# B&R Automation Studio project SuperTrakProject (part 2)

#### Main.st
```iecst
(***************************************************************************************
 * STSection task
 *
 * This task provides a state machine for controlling and monitoring
 * SuperTrak Sections. This task can be interfaced with via gSuperTrak.Sections
 *
 * File: STSection.st
 * Created: 2024-08-15
 *
 * Authors:
 *  Marcus Mangel, B&R Industrial Automation
 *  Tyler Matijevich, B&R Industrial Automation
 *
***************************************************************************************)

PROGRAM _CYCLIC

    // Read global inputs
    Interface.Cmd := gSuperTrak.Sections.Cmd;

    // Initialize common statuses, assume true/false then disqualify
    Interface.Status.Active := TRUE;
    Interface.Status.Error := FALSE;
	Interface.Status.SectionError := 0;
	Interface.Status.SectionWarning := 0;

    FOR Index := 1 TO ST_SECTION_MAX DO
        ControlSection[Index].StLink := ADR(gSTSystemLink);
        ControlSection[Index].Section := Index;
        // There are no function block parameters, use common address
        ControlSection[Index].Parameters := ADR(SectionParameters[Index]);
        // Enable all function blocks one the System is Active
        ControlSection[Index].Enable := gSuperTrak.System.Status.Active;
        // Enable each section
        ControlSection[Index].EnableSection := Interface.Cmd.PowerSection[Index] AND ControlSection[Index].MotorPowerOn AND NOT ControlSection[Index].Error;
        // Reset all function blocks
        ControlSection[Index].ErrorReset := gSuperTrak.System.Cmd.Reset AND ControlSection[Index].Error;
        ControlSection[Index]();

        // All sections must be active
        IF ControlSection[Index].Active = FALSE THEN
            Interface.Status.Active := FALSE;
        END_IF
        // Error if any section has error
        IF ControlSection[Index].Error THEN
            Interface.Status.Error := TRUE;
            Interface.Status.StatusID := ControlSection[Index].StatusID;
        END_IF
        IF ControlSection[Index].Info.SuperTrak.SectionFaultActive THEN
            Interface.Status.SectionError := Index;
		END_IF;
		IF ControlSection[Index].Info.SuperTrak.SectionWarningActive THEN
			Interface.Status.SectionWarning:= Index;
        END_IF;

        // Log errors only when that error first occurs
        r_trig_SectionFBError[Index](CLK := ControlSection[Index].Error);
        r_trig_SectionWarning[Index](CLK := ControlSection[Index].Info.SuperTrak.SectionWarningActive);
        r_trig_SectionFault[Index](CLK := ControlSection[Index].Info.SuperTrak.SectionFaultActive);

        IF r_trig_SectionFBError[Index].Q THEN
            brsmemset(ADR(UserLogArguments), 0, SIZEOF(UserLogArguments));
            UserLogArguments.i[0] := Index;
            UserLogArguments.i[1] := ControlSection[Index].StatusID;
            UserLogEventText('$$arlogusr', -536869812, 0, '', '%i %i', UserLogArguments);
        END_IF;
        IF r_trig_SectionWarning[Index].Q THEN
            brsmemset(ADR(UserLogArguments), 0, SIZEOF(UserLogArguments));
            UserLogArguments.i[0] := Index;
            UserLogArguments.i[1] := ControlSection[Index].Info.SuperTrak.SectionWarningBits;
            UserLogEventText('$$arlogusr', -1610609636, 0, '', '%i %i', UserLogArguments);
        END_IF;
        IF r_trig_SectionFault[Index].Q THEN
            brsmemset(ADR(UserLogArguments), 0, SIZEOF(UserLogArguments));
            UserLogArguments.i[0] := Index;
            UserLogArguments.i[1] := ControlSection[Index].Info.SuperTrak.SectionFaultBits;
            UserLogEventText('$$arlogusr', -536869810, 0, '', '%i %i', UserLogArguments);
        END_IF;

        // Read other statuses
        Interface.Info[Index].SectionEnabled := ControlSection[Index].SectionEnabled;
        Interface.Info[Index].UnrecognizedShuttles := ControlSection[Index].UnrecognizedPallets;
        Interface.Info[Index].MotorPowerOn := ControlSection[Index].MotorPowerOn;
        Interface.Info[Index].ShuttlesRecovering := ControlSection[Index].PalletsRecovering;
        Interface.Info[Index].LocatingShuttles := ControlSection[Index].LocatingPallets;
        Interface.Info[Index].DisabledExternally := ControlSection[Index].DisabledExternally;
        Interface.Info[Index].WarningPresent := ControlSection[Index].Info.SuperTrak.SectionWarningActive;
        Interface.Info[Index].Warnings := ControlSection[Index].Info.SuperTrak.SectionWarningBits;
        Interface.Info[Index].FaultPresent := ControlSection[Index].Info.SuperTrak.SectionFaultActive;
        Interface.Info[Index].Faults := ControlSection[Index].Info.SuperTrak.SectionFaultBits;
    END_FOR

    // Write global outputs
	gSuperTrak.Sections.Status := Interface.Status;
	gSuperTrak.Sections.Info := Interface.Info;

END_PROGRAM
```

### Package Logical/Source/STMgr/STTarget - StCom target control

### STTarget.typ - Global types
```iecst
(***************************************************************************************
 * Global STTarget data types
 *
 * These structures allow any program (task) to interface with the STTarget task
 *
 * File: STTarget.typ
 * Created: 2024-08-15
 *
 * Authors:
 *  Marcus Mangel, B&R Industrial Automation
 *
****************************************************************************************)

TYPE
    STTargetInterfaceType :     STRUCT  (*Target control interface*)
        Cmd : STTargetCommandType; (*Target release and set shuttle parameter commands*)
        Par : STTargetParType; (*Target control parameters*)
        Status : STTargetStatusType; (*Target status structure*)
    END_STRUCT;
    STTargetCommandType :     STRUCT  (*Target release and set shuttle parameter commands*)
        Release : STReleaseCommandType; (*Target release commands*)
        SetShuttleID : BOOL; (*Set the ID of the shuttle at the target*)
    END_STRUCT;
    STTargetParType :     STRUCT  (*Target control parameters*)
        Release : STReleaseParameterType; (*Target release parameters*)
        SetShuttleID : USINT; (*Set the current shuttle's ID to this when commanded*)
    END_STRUCT;
    STTargetStatusType :     STRUCT  (*Target status structure*)
        Active : BOOL; (*Target Control function block is active*)
        Error : BOOL; (*Target Control function block is reporting an error*)
        StatusID : DINT; (*Status ID from the Target Control function block*)
        ShuttlePresent : BOOL; (*A shuttle has arrived, has entered the in-position window, and has not yet been released*)
        ShuttleInPosition : BOOL; (*A shuttle is currently within the in-position window*)
        ShuttlePreArrival : BOOL; (*A shuttle is expected to arrive at the stop within the configured time*)
        ShuttleOverTarget : BOOL; (*A shuttle's shelf is over the target, only reported if configured*)
        ShuttleOffsetIndex : USINT; (*Offset-Table index applied to the shuttle at the target*)
        ShuttleID : USINT; (*ID of shuttle present at target, pallet over target (if configured), or pallet from pre-arrival notification (if configured)*)
        ShuttleReleased : BOOL; (*(Derived) Release command acknowledged. True until release command is reset*)
        ShuttleCount : USINT; (*(Derived) Number of shuttles destined for target*)
        Section : USINT; (*(Par 1650) Target section number*)
        PositionMicrons : DINT; (*(Par 1651) [um] Target section position in microns*)
        Position : REAL; (*(Par 1651) [mm] Target section position*)
        ShuttleIDSet : BOOL; (*The Shuttle ID was successfully set. True until the command is reset*)
    END_STRUCT;
END_TYPE
```

### Program Logical/Source/STMgr/STTarget/STTarget (IEC) - StCom target control

#### Main.st - Init, cyclic, exit code
```iecst
(***************************************************************************************
 * STTarget task
 *
 * This task provides a state machine for controlling and monitoring
 * SuperTrak Targets. This task can be interfaced with via gSuperTrak.Target[Target #]
 * where "Target #" is an array value indexed starting at 1 (see: Trakmaster targets)
 *
 * File: STTarget.st
 * Created: 2024-08-15
 *
 * Authors:
 *  Marcus Mangel, B&R Industrial Automation
 *
***************************************************************************************)

PROGRAM _CYCLIC

    // Get data for all targets when the system is active
    IF gSuperTrak.System.Status.Active THEN
        SuperTrakServChanRead(0, 1650, 0, 256, ADR(Sections), SIZEOF(Sections));
        SuperTrakServChanRead(0, 1651, 0, 256, ADR(Positions), SIZEOF(Positions));
    END_IF;

    FOR Index := 1 TO ST_TARGET_MAX DO
        // Read global inputs
        Interface[Index].Cmd := gSuperTrak.Target[Index].Cmd;
        Interface[Index].Par := gSuperTrak.Target[Index].Par;

        // Link parameters
        TargetParameters[Index].AdvancedReleaseConfig.DestinationTarget := Interface[Index].Par.Release.DestinationTarget;
        TargetParameters[Index].AdvancedReleaseConfig.IncrementalOffset := LIMIT(-500.0, Interface[Index].Par.Release.IncrementalOffset, 500.0);
        TargetParameters[Index].AdvancedReleaseConfig.TargetOffset := LIMIT(-500.0, Interface[Index].Par.Release.TargetOffset, 500.0);
        TargetParameters[Index].AdvancedReleaseConfig.Direction := Interface[Index].Par.Release.Direction;
        TargetParameters[Index].PalletConfig.Motion.Acceleration := REAL_TO_UINT(LIMIT(1, Interface[Index].Par.Release.Acceleration, 60) * METERS_TO_MILLIMETERS);
        TargetParameters[Index].PalletConfig.Motion.Velocity := REAL_TO_UINT(LIMIT(10, Interface[Index].Par.Release.Velocity, 4000));
        TargetParameters[Index].PalletConfig.ID := Interface[Index].Par.SetShuttleID;

        // StTargetExt function block inputs
        ControlTarget[Index].StLink := ADR(gSTSystemLink);
        ControlTarget[Index].Enable := gSuperTrak.System.Status.Active;
        ControlTarget[Index].ErrorReset := gSuperTrak.System.Cmd.Reset AND ControlTarget[Index].Error;
        ControlTarget[Index].Parameters := ADR(TargetParameters[Index]);
        ControlTarget[Index].Target := Index;

        // If the function block errored out, reset it's commands to prevent an error loop
        IF ControlTarget[Index].ErrorReset THEN
            ControlTarget[Index].ReleaseToTarget := FALSE;
            ControlTarget[Index].ReleaseToOffset := FALSE;
            ControlTarget[Index].IncrementOffset := FALSE;
	        TargetControlState[Index] := TARGET_STATE_WAIT_FOR_CMD_RESET;
        END_IF;

        CASE TargetControlState[Index] OF
            TARGET_STATE_WAIT_FOR_SHUTTLE:
                IF ControlTarget[Index].PalletPresent THEN
                    TargetControlState[Index] := TARGET_STATE_SHUTTLE_PRESENT;
                END_IF;

            TARGET_STATE_SHUTTLE_PRESENT:
                IF Interface[Index].Cmd.SetShuttleID THEN
                    TargetControlState[Index] := TARGET_STATE_SET_SHUTTLE_ID;
                ELSIF Interface[Index].Cmd.Release.ReleaseToTarget OR Interface[Index].Cmd.Release.ReleaseToOffset OR Interface[Index].Cmd.Release.IncrementOffset THEN
                    TargetControlState[Index] := TARGET_STATE_SET_MOTION_PARS;
                END_IF;

            TARGET_STATE_SET_SHUTTLE_ID:
                ControlTarget[Index].SetPalletID := TRUE;
                IF ControlTarget[Index].CommandDone THEN
                    ControlTarget[Index].SetPalletID := FALSE;
                    Interface[Index].Status.ShuttleIDSet := TRUE;
                    TargetControlState[Index] := TARGET_STATE_WAIT_FOR_CMD_RESET;
                END_IF;

            TARGET_STATE_SET_MOTION_PARS:
                ControlTarget[Index].SetPalletMotionPar := TRUE;
                IF ControlTarget[Index].CommandDone THEN
                    ControlTarget[Index].SetPalletMotionPar := FALSE;
                    TargetControlState[Index] := TARGET_STATE_RELEASE_SHUTTLE;
                END_IF;

            TARGET_STATE_RELEASE_SHUTTLE:
                ControlTarget[Index].ReleaseToTarget := Interface[Index].Cmd.Release.ReleaseToTarget; // Trust that the user won't set more than
                ControlTarget[Index].ReleaseToOffset := Interface[Index].Cmd.Release.ReleaseToOffset; // one of these at the same time
                ControlTarget[Index].IncrementOffset := Interface[Index].Cmd.Release.IncrementOffset; // Not sure what would happen in that case
                TargetControlState[Index] := TARGET_STATE_WAIT_FOR_RELEASE;

            TARGET_STATE_WAIT_FOR_RELEASE:
                IF NOT ControlTarget[Index].PalletPresent THEN
                    ControlTarget[Index].ReleaseToTarget := FALSE;
                    ControlTarget[Index].ReleaseToOffset := FALSE;
                    ControlTarget[Index].IncrementOffset := FALSE;
                    Interface[Index].Status.ShuttleReleased := TRUE;
                    TargetControlState[Index] := TARGET_STATE_WAIT_FOR_CMD_RESET;
                END_IF;

            TARGET_STATE_WAIT_FOR_CMD_RESET:
                IF NOT (Interface[Index].Cmd.SetShuttleID OR Interface[Index].Cmd.Release.ReleaseToTarget
                    OR Interface[Index].Cmd.Release.ReleaseToOffset OR Interface[Index].Cmd.Release.IncrementOffset) THEN
                    Interface[Index].Status.ShuttleReleased := FALSE;
                    Interface[Index].Status.ShuttleIDSet := FALSE; // Reset all "Command Done" Statuses
                    TargetControlState[Index] := TARGET_STATE_WAIT_FOR_SHUTTLE;
                END_IF;
        END_CASE;

        // Call StTargetExt function block
        ControlTarget[Index]();

        // Read StTargetExt function block outputs
        Interface[Index].Status.Active := ControlTarget[Index].Active;
        Interface[Index].Status.Error := ControlTarget[Index].Error;
        Interface[Index].Status.StatusID := ControlTarget[Index].StatusID;
        Interface[Index].Status.ShuttleID := ControlTarget[Index].PalletID;
        Interface[Index].Status.ShuttleOffsetIndex := ControlTarget[Index].PalletOffsetIdx;
        Interface[Index].Status.ShuttlePresent := ControlTarget[Index].PalletPresent;
        Interface[Index].Status.ShuttleInPosition := ControlTarget[Index].PalletInPosition;
        Interface[Index].Status.ShuttlePreArrival := ControlTarget[Index].PalletPreArrival;
        Interface[Index].Status.ShuttleOverTarget := ControlTarget[Index].PalletOverTarget;
        Interface[Index].Status.Section := UINT_TO_USINT(Sections[Index]);
        Interface[Index].Status.PositionMicrons := Positions[Index];
        Interface[Index].Status.Position := DINT_TO_REAL(Interface[Index].Status.PositionMicrons)/1000.0;

        // Log errors only when that error first occurs
        r_trig_TargetFBError[Index](CLK := ControlTarget[Index].Error);

        IF r_trig_TargetFBError[Index].Q THEN
            brsmemset(ADR(UserLogArguments), 0, SIZEOF(UserLogArguments));
            UserLogArguments.i[0] := Index;
            UserLogArguments.i[1] := ControlTarget[Index].StatusID;
            UserLogEventText('$$arlogusr', -536869712, 0, '', '%i %i', UserLogArguments);
        END_IF;

        // Check for release commands and update ShuttleCount status
        r_trig_ShuttleRelease[Index].CLK := (Interface[Index].Cmd.Release.ReleaseToTarget
        OR Interface[Index].Cmd.Release.ReleaseToOffset OR Interface[Index].Cmd.Release.IncrementOffset);
        r_trig_ShuttleRelease[Index]();

        IF r_trig_ShuttleRelease[Index].Q THEN
            // Decrement this target's shuttle count
            IF Interface[Index].Status.ShuttleCount > 0 THEN
                Interface[Index].Status.ShuttleCount := Interface[Index].Status.ShuttleCount - 1;
            END_IF;
            // Increment destination target's shuttle count
            IF Interface[Index].Par.Release.DestinationTarget > 0 AND Interface[Index].Par.Release.DestinationTarget <= ST_TARGET_MAX THEN
                Interface[Interface[Index].Par.Release.DestinationTarget].Status.ShuttleCount :=
                Interface[Interface[Index].Par.Release.DestinationTarget].Status.ShuttleCount + 1;
            END_IF;
        END_IF;

        // Write global outputs
        gSuperTrak.Target[Index].Status := Interface[Index].Status;
    END_FOR

END_PROGRAM
```

#### Types.typ
```iecst
(***************************************************************************************
 * STTarget task local data types
 *
 * These structures and enumerations are local to the STTarget task
 *
 * File: STTarget/Types.typ
 * Created: 2024-08-15
 *
 * Authors:
 *  Marcus Mangel, B&R Industrial Automation
 *
***************************************************************************************)
TYPE
	TargetControlState_enum :
		( (*Shuttle release state machine*)
		TARGET_STATE_WAIT_FOR_SHUTTLE, (*Wait for a shuttle to arrive at the target*)
		TARGET_STATE_SHUTTLE_PRESENT, (*A shuttle is at the target and ready for commands*)
		TARGET_STATE_SET_SHUTTLE_ID, (*Set the ID of the shuttle that is currently at the target*)
		TARGET_STATE_SET_MOTION_PARS, (*Set the shutte at target's motion parameters*)
		TARGET_STATE_RELEASE_SHUTTLE, (*Release the shuttle currently at the target*)
		TARGET_STATE_WAIT_FOR_RELEASE, (*Wait for the release to complete*)
		TARGET_STATE_WAIT_FOR_CMD_RESET (*Wait for the caller to reset all commands*)
		);
END_TYPE
```

#### Variables.var - Local variables
```iecst
(***************************************************************************************
 * STTarget task local variables
 *
 * These variables are local to the STTarget task
 *
 * File: STTarget/Variables.var
 * Created: 2024-08-15
 *
 * Authors:
 *  Marcus Mangel, B&R Industrial Automation
 *
***************************************************************************************)
VAR
	Interface : ARRAY[1..ST_TARGET_MAX] OF STTargetInterfaceType; (*Local copy of gSuperTrak.Target*)
	TargetControlState : ARRAY[1..ST_TARGET_MAX] OF TargetControlState_enum; (*Shuttle release state machine*)
	TargetParameters : ARRAY[1..ST_TARGET_MAX] OF StTargetExtParType; (*Target control parameters*)
	ControlTarget : ARRAY[1..ST_TARGET_MAX] OF StTargetExt; (*Target control function block*)
	Sections : ARRAY[0..255] OF UINT; (*All target sections*)
	Positions : ARRAY[0..255] OF DINT; (*All target positions*)
	Index : USINT; (*FOR loop index*)
	r_trig_ShuttleRelease : ARRAY[1..ST_TARGET_MAX] OF R_TRIG; (*Rising edge trigger of any Release command*)
	UserLogArguments : UserLogFormatType; (*Arguments used in Logger messages (UserLog library)*)
	r_trig_TargetFBError : ARRAY[1..ST_TARGET_MAX] OF R_TRIG; (*Rising edge trigger for ControlTarget.Error*)
END_VAR
```

### Package Logical/Source/STMgr/STShuttle - StCom shuttle (pallet) control

### STShuttle.typ - Global types
```iecst
(***************************************************************************************
 * Global STShuttle data types
 *
 * These structures allow any program (task) to interface with the STShuttle task
 *
 * File: STShuttle.typ
 * Created: 2024-08-15
 *
 * Authors:
 *  Marcus Mangel, B&R Industrial Automation
 *
****************************************************************************************)

TYPE
    STShuttleInterfaceType :     STRUCT  (*Shuttle interface structure*)
        Cmd : STReleaseCommandType; (*Shuttle release commands*)
        Status : STShuttleStatusType; (*Shuttle status information*)
        Par : STReleaseParameterType; (*Shuttle release parameters*)
    END_STRUCT;
    STShuttleStatusType :     STRUCT  (*Shuttle status structure*)
        Active : BOOL; (*Shuttle Control function block is active*)
        Error : BOOL; (*Shuttle Control function block is reporting an error*)
        StatusID : DINT; (*Status ID from the Shuttle Control function block*)
        ShuttleID : USINT; (*(StPalletStatusBits_e) ID Number assigned to the shuttle*)
        Present : BOOL; (*(StPalletStatusBits_e) Present on system*)
        Recovering : BOOL; (*(StPalletStatusBits_e) Will recover or recovering to last controlled position*)
        AtTarget : BOOL; (*(StPalletStatusBits_e) Arrived at target, in position, not yet released*)
        InPosition : BOOL; (*(StPalletStatusBits_e) Within in-position window*)
        ServoEnabled : BOOL; (*(StPalletStatusBits_e) Control enabled*)
        Initializing : BOOL; (*(StPalletStatusBits_e) Moving to load target*)
        Lost : BOOL; (*(StPalletStatusBits_e) Position feedback lost*)
        ControlMode : USINT; (*(SuperTrakPalletInfo_t) Pallet control mode, see SuperTrak library*)
        Section : USINT; (*(SuperTrakPalletInfo_t or Par 1307) Current section number*)
        PositionMicrons : DINT; (*(SuperTrakPalletInfo_t or Par 1310) [um] Current section position in microns*)
        Position : REAL; (*(SuperTrakPalletInfo_t or Par 1310) [mm] Current section position*)
        Velocity : REAL; (*(Par 1314) [mm/s] Current velocity*)
        DestinationTarget : USINT; (*(Par 1339) Destination target*)
        SetSection : USINT; (*(Par 1306) Section number setpoint*)
        SetPositionMicrons : DINT; (*(Par 1311) [um] Integer section position setpoint in microns*)
        SetPosition : REAL; (*(Par 1311) [mm] Section position setpoint*)
        SetVelocity : REAL; (*(Par 1313) [mm/s] Velocity setpoint*)
        SetAcceleration : REAL; (*(Par 1312) [m/s^2] Acceleration setpoint (raw value is mm/s^2!]*)
        ShuttleReleased : BOOL; (*(Derived) Release command acknowledged. True until release command is reset*)
    END_STRUCT;
END_TYPE
```

### Program Logical/Source/STMgr/STShuttle/STShuttle (IEC) - StCom shuttle control

#### Types.typ
```iecst
(***************************************************************************************
 * STShuttle task local data types
 *
 * These structures and enumerations are local to the STShuttle task
 *
 * File: STShuttle/Types.typ
 * Created: 2024-08-15
 *
 * Authors:
 *  Marcus Mangel, B&R Industrial Automation
 *
***************************************************************************************)
TYPE
	ShuttleControlState_enum :
		( (*State machine for Shuttle control*)
		SHUTTLE_STATE_WAIT_FOR_COMMAND, (*Wait for a command*)
		SHUTTLE_STATE_SET_MOTION_PARS, (*Set the shuttle's velocity and acceleration*)
		SHUTTLE_STATE_RELEASE_SHUTTLE, (*Give the shuttle a release command*)
		SHUTTLE_STATE_WAIT_FOR_CMD_RESET (*Wait for interface commands to be reset by the caller*)
		);
END_TYPE
```

#### Variables.var
```iecst
(***************************************************************************************
 * STShuttle task local variables
 *
 * These variables are local to the STShuttle task
 *
 * File: STShuttle/Variables.var
 * Created: 2024-08-15
 *
 * Authors:
 *  Marcus Mangel, B&R Industrial Automation
 *
***************************************************************************************)
VAR
	Interface : ARRAY[1..ST_SHUTTLE_MAX] OF STShuttleInterfaceType; (*Local copy of gSuperTrak.Shuttle*)
	ShuttleControlState : ARRAY[1..ST_SHUTTLE_MAX] OF ShuttleControlState_enum; (*Shuttle release state machine*)
	ShuttleParameters : ARRAY[1..ST_SHUTTLE_MAX] OF StPalletParType; (*Shuttle control parameters*)
	ControlShuttle : ARRAY[1..ST_SHUTTLE_MAX] OF StPallet; (*Shuttle control function block*)
	ShuttleInfo : ARRAY[1..ST_SHUTTLE_MAX] OF SuperTrakPalletInfo_t; (*Shuttle status information*)
	ActualVelocity : ARRAY[0..255] OF INT; (*Actual Velocity information for all shuttles*)
	DestinationTarget : ARRAY[0..255] OF UINT; (*Destination Target information for all shuttles*)
	SectionSetpoint : ARRAY[0..255] OF UINT; (*Section Setpoint information for all shuttles*)
	PositionSetpoint : ARRAY[0..255] OF DINT; (*Position Setpoint information for all shuttles*)
	VelocitySetpoint : ARRAY[0..255] OF REAL; (*Velocity Setpoint information for all shuttles*)
	AccelerationSetpoint : ARRAY[0..255] OF REAL; (*Acceleration Setpoint information for all shuttles*)
	Index : USINT; (*FOR Loop index*)
	r_trig_ShuttleRelease : ARRAY[1..ST_SHUTTLE_MAX] OF R_TRIG; (*Rising edge trigger of any Release command*)
	ShuttleAtTarget : USINT; (*Used during release to check the Target a Shuttle is currently at*)
	TargetIndex : USINT; (*FOR loop index*)
	UserLogArguments : UserLogFormatType; (*Arguments used in Logger messages (UserLog library)*)
	r_trig_ShuttleFBError : ARRAY[1..ST_SHUTTLE_MAX] OF R_TRIG; (*Rising edge trigger for ControlShuttle.Error*)
END_VAR
```

#### Main.st
```iecst
(*******************************************************************************************
 * STShuttle task
 *
 * This task provides a state machine for controlling and monitoring
 * SuperTrak Shuttles. This task can be interfaced with via gSuperTrak.Shuttle[Shuttle #]
 * where "Shuttle #" is an array value indexed starting at 1 (see: Trakmaster shuttles)
 *
 * File: STShuttle.st
 * Created: 2024-08-15
 *
 * Authors:
 *  Marcus Mangel, B&R Industrial Automation
 *
*******************************************************************************************)

PROGRAM _CYCLIC

    // Get data for all shuttles when the system is active
    IF gSuperTrak.System.Status.Active THEN
        // Call SuperTrakGetPalletInfo function
        SuperTrakGetPalletInfo(ADR(ShuttleInfo), SIZEOF(ShuttleInfo)/SIZEOF(ShuttleInfo[1]), FALSE); // FALSE - Return actual positions of shuttles

        // Read additional parameters via the Service Channel
        SuperTrakServChanRead(0, 1314, 0, 256, ADR(ActualVelocity), SIZEOF(ActualVelocity));
        SuperTrakServChanRead(0, 1339, 0, 256, ADR(DestinationTarget), SIZEOF(DestinationTarget));
        SuperTrakServChanRead(0, 1306, 0, 256, ADR(SectionSetpoint), SIZEOF(SectionSetpoint));
        SuperTrakServChanRead(0, 1311, 0, 256, ADR(PositionSetpoint), SIZEOF(PositionSetpoint));
        SuperTrakServChanRead(0, 1313, 0, 256, ADR(VelocitySetpoint), SIZEOF(VelocitySetpoint));
        SuperTrakServChanRead(0, 1312, 0, 256, ADR(AccelerationSetpoint), SIZEOF(AccelerationSetpoint));
    END_IF;

    FOR Index := 1 TO ST_SHUTTLE_MAX DO
        // Read global inputs
        Interface[Index].Cmd := gSuperTrak.Shuttle[Index].Cmd;
        Interface[Index].Par := gSuperTrak.Shuttle[Index].Par;

        // Link parameters
        ShuttleParameters[Index].AdvancedReleaseConfig.DestinationTarget := Interface[Index].Par.DestinationTarget;
        ShuttleParameters[Index].AdvancedReleaseConfig.IncrementalOffset := LIMIT(-500.0, Interface[Index].Par.IncrementalOffset, 500.0);
        ShuttleParameters[Index].AdvancedReleaseConfig.TargetOffset := LIMIT(-500.0, Interface[Index].Par.TargetOffset, 500.0);
        ShuttleParameters[Index].AdvancedReleaseConfig.Direction := Interface[Index].Par.Direction;
        ShuttleParameters[Index].PalletConfig.Motion.Acceleration := REAL_TO_UINT(LIMIT(1, Interface[Index].Par.Acceleration, 60) * METERS_TO_MILLIMETERS);
        ShuttleParameters[Index].PalletConfig.Motion.Velocity := REAL_TO_UINT(LIMIT(10, Interface[Index].Par.Velocity, 4000));

        // StShuttleExt function block inputs
        ControlShuttle[Index].StLink := ADR(gSTSystemLink);
        ControlShuttle[Index].Enable := gSuperTrak.System.Status.Active;
        ControlShuttle[Index].ErrorReset := gSuperTrak.System.Cmd.Reset AND ControlShuttle[Index].Error;
        ControlShuttle[Index].Parameters := ADR(ShuttleParameters[Index]);
        ControlShuttle[Index].PalletID := Index;

        // If the function block errored out, reset it's commands to prevent an error loop
        IF ControlShuttle[Index].ErrorReset THEN
            ControlShuttle[Index].ReleaseToTarget := FALSE;
            ControlShuttle[Index].ReleaseToOffset := FALSE;
            ControlShuttle[Index].IncrementOffset := FALSE;
            ShuttleControlState[Index] := SHUTTLE_STATE_WAIT_FOR_CMD_RESET;
        END_IF;

        CASE ShuttleControlState[Index] OF
            SHUTTLE_STATE_WAIT_FOR_COMMAND:
                IF Interface[Index].Cmd.ReleaseToTarget OR Interface[Index].Cmd.ReleaseToOffset OR Interface[Index].Cmd.IncrementOffset THEN
                    ShuttleControlState[Index] := SHUTTLE_STATE_SET_MOTION_PARS;
                END_IF;

            SHUTTLE_STATE_SET_MOTION_PARS:
                ControlShuttle[Index].SetPalletMotionPar := TRUE;
                IF ControlShuttle[Index].CommandDone THEN
                    ControlShuttle[Index].SetPalletMotionPar := FALSE;
                    ShuttleControlState[Index] := SHUTTLE_STATE_RELEASE_SHUTTLE;
                END_IF;

            SHUTTLE_STATE_RELEASE_SHUTTLE:
                ControlShuttle[Index].ReleaseToTarget := Interface[Index].Cmd.ReleaseToTarget;
                ControlShuttle[Index].ReleaseToOffset := Interface[Index].Cmd.ReleaseToOffset;
                ControlShuttle[Index].IncrementOffset := Interface[Index].Cmd.IncrementOffset;
                Interface[Index].Status.ShuttleReleased := TRUE;
                ShuttleControlState[Index] := SHUTTLE_STATE_WAIT_FOR_CMD_RESET;

            SHUTTLE_STATE_WAIT_FOR_CMD_RESET:
                IF NOT(Interface[Index].Cmd.ReleaseToTarget OR Interface[Index].Cmd.ReleaseToOffset OR Interface[Index].Cmd.IncrementOffset) THEN
                    Interface[Index].Status.ShuttleReleased := FALSE;
                    ControlShuttle[Index].ReleaseToTarget := FALSE;
                    ControlShuttle[Index].ReleaseToOffset := FALSE;
                    ControlShuttle[Index].IncrementOffset := FALSE;
                    ShuttleControlState[Index] := SHUTTLE_STATE_WAIT_FOR_COMMAND;
                END_IF;
        END_CASE;

        // Call StShuttleExt function block
        ControlShuttle[Index]();

        // Read function outputs
        Interface[Index].Status.Active := ControlShuttle[Index].Active;
        Interface[Index].Status.Error := ControlShuttle[Index].Error;
        Interface[Index].Status.StatusID := ControlShuttle[Index].StatusID;
        Interface[Index].Status.ShuttleID := ShuttleInfo[Index].palletID;
        Interface[Index].Status.Present := ShuttleInfo[Index].status.stPALLET_PRESENT;
        Interface[Index].Status.Recovering := ShuttleInfo[Index].status.stPALLET_RECOVERING;
        Interface[Index].Status.AtTarget := ShuttleInfo[Index].status.stPALLET_AT_TARGET;
        Interface[Index].Status.InPosition := ShuttleInfo[Index].status.stPALLET_IN_POSITION;
        Interface[Index].Status.ServoEnabled := ShuttleInfo[Index].status.stPALLET_SERVO_ENABLED;
        Interface[Index].Status.Initializing := ShuttleInfo[Index].status.stPALLET_INITIALIZING;
        Interface[Index].Status.Lost := ShuttleInfo[Index].status.stPALLET_LOST;
        Interface[Index].Status.ControlMode := ShuttleInfo[Index].controlMode;
        Interface[Index].Status.Section := ShuttleInfo[Index].section;
        Interface[Index].Status.PositionMicrons := ShuttleInfo[Index].position;
        Interface[Index].Status.Position := DINT_TO_REAL(Interface[Index].Status.PositionMicrons)/1000.0;
        Interface[Index].Status.Velocity := INT_TO_REAL(ActualVelocity[Index]);
        Interface[Index].Status.DestinationTarget := UINT_TO_USINT(DestinationTarget[Index]);
        Interface[Index].Status.SetSection := UINT_TO_USINT(SectionSetpoint[Index]);
        Interface[Index].Status.SetPositionMicrons := PositionSetpoint[Index];
        Interface[Index].Status.SetPosition := DINT_TO_REAL(Interface[Index].Status.SetPositionMicrons)/1000.0;
        Interface[Index].Status.SetVelocity := VelocitySetpoint[Index];
        Interface[Index].Status.SetAcceleration := AccelerationSetpoint[Index] / METERS_TO_MILLIMETERS;

        // Log errors only when that error first occurs
        r_trig_ShuttleFBError[Index](CLK := ControlShuttle[Index].Error);

        IF r_trig_ShuttleFBError[Index].Q THEN
            brsmemset(ADR(UserLogArguments), 0, SIZEOF(UserLogArguments));
            UserLogArguments.i[0] := Index;
            UserLogArguments.i[1] := ControlShuttle[Index].StatusID;
            UserLogEventText('$$arlogusr', -536869612, 0, '', '%i %i', UserLogArguments);
        END_IF;

        // Check for release commands and update Target ShuttleCount statuses
        r_trig_ShuttleRelease[Index].CLK := (Interface[Index].Cmd.ReleaseToTarget OR Interface[Index].Cmd.ReleaseToOffset OR Interface[Index].Cmd.IncrementOffset);
        r_trig_ShuttleRelease[Index]();

        IF r_trig_ShuttleRelease[Index].Q THEN
            // Decrement current target's shuttle count (if shuttle is currently at a target)
            IF Interface[Index].Status.AtTarget THEN
                ShuttleAtTarget := 0;
                FOR TargetIndex := 1 TO ST_TARGET_MAX DO
                    IF gSuperTrak.Target[TargetIndex].Status.ShuttlePresent AND gSuperTrak.Target[TargetIndex].Status.ShuttleID = Index THEN
                        ShuttleAtTarget := TargetIndex;
                        EXIT;
                    END_IF;
                END_FOR;

                IF ShuttleAtTarget > 0 AND ShuttleAtTarget <= ST_TARGET_MAX THEN
                    IF gSuperTrak.Target[ShuttleAtTarget].Status.ShuttleCount > 0 THEN
                        gSuperTrak.Target[ShuttleAtTarget].Status.ShuttleCount := gSuperTrak.Target[ShuttleAtTarget].Status.ShuttleCount - 1;
                    END_IF;
                END_IF;
            END_IF;
            // Increment destination target's shuttle count
            IF gSuperTrak.Shuttle[Index].Par.DestinationTarget > 0 AND gSuperTrak.Shuttle[Index].Par.DestinationTarget <= ST_TARGET_MAX THEN
                gSuperTrak.Target[gSuperTrak.Shuttle[Index].Par.DestinationTarget].Status.ShuttleCount :=
                gSuperTrak.Target[gSuperTrak.Shuttle[Index].Par.DestinationTarget].Status.ShuttleCount + 1;
            END_IF;
        END_IF;

        // Write global outputs
        gSuperTrak.Shuttle[Index].Status := Interface[Index].Status;
    END_FOR

END_PROGRAM
```

### Package Logical/Source/EthIP - EtherNet/IP communication

### Program Logical/Source/EthIP/EipComm (IEC) - EtherNet/IP communication task

#### Main.st - Init, cyclic, exit code
```iecst
(***************************************************************************************
 * EipComm task
 *
 * This task handles Ethernet/IP Communication. It is only used if the SuperTrak will
 * be controlled by another PLC via EtherNet/IP. This task exchanges Ethernet/IP
 * data with the gSuperTrak structure.
 *
 * The data that will be exchanged is defined in the ethIPcon.dat file
 *
 * This is meant to be a starting point, but more data may need to be communicated
 * depending on the application
 *
 * File: EipComm.st
 * Created: 2025-03-12
 *
 * Authors:
 *  Marcus Mangel, B&R Industrial Automation
 *
***************************************************************************************)

PROGRAM _INIT

    // Set TaskIsSimulated initially based on ARSim usage
    // This can be set False if a real Ethernet/IP connection will be established to ARSim
    TaskIsSimulated := DiagCpuIsARsim();

    // Make sure this compiles
    StationStatus;

    // Initialize Ethernet IP communication
    // This must be done in the INIT program
    fb_EIPInit.enable := TRUE;
    fb_EIPInit.pconfig := ADR('ethIPcon');
    fb_EIPInit();
    InitExitStatus := fb_EIPInit.extstatus;

    IF fb_EIPInit.status = 0 THEN
        Initialized := TRUE;
        InitHandle := fb_EIPInit.handle;
        brsmemset(ADR(UserLogArguments), 0, SIZEOF(UserLogArguments));
        UserLogCustom('$$arlogusr', USERLOG_SEVERITY_INFORMATION, 1, 30, 0, '', 'EtherNet/IP data object initialized successfully', UserLogArguments);
    ELSE
        Initialized := FALSE;
        InitHandle := 0;
        brsmemset(ADR(UserLogArguments), 0, SIZEOF(UserLogArguments));
        brsstrcpy(ADR(UserLogArguments.s[0]), ADR(fb_EIPInit.extstatus));
        UserLogCustom('$$arlogusr', USERLOG_SEVERITY_ERROR, 1, 10, 0, '', 'EtherNet/IP data object initialization failed! Status: %s', UserLogArguments);
        CommState := COMM_STATE_ERROR;
    END_IF;

END_PROGRAM

PROGRAM _CYCLIC

    (** !!! Disable this task in the Software Configuration if it is not used!
         This prevents data from being overwritten !!! **)

    // If this task is running, tell the Main task that control is being done externally
	gUseExternalControl := TRUE;

    // Check for errors
    // Function Block may return ERR_FUB_ENABLE_FALSE or ERR_FUB_BUSY during normal operation
    // Any other nonzero status is an error
    IF EDGEPOS((fb_EIPCyclic.status <> 0) AND (fb_EIPCyclic.status <> ERR_FUB_ENABLE_FALSE) AND (fb_EIPCyclic.status <> ERR_FUB_BUSY)) THEN
        brsmemset(ADR(UserLogArguments), 0, SIZEOF(UserLogArguments));
        UserLogArguments.i[0] := fb_EIPCyclic.status;
        UserLogCustom('$$arlogusr', USERLOG_SEVERITY_ERROR, 1, 11, 0, '', 'EtherNet/IP communication error: %i', UserLogArguments);
        CommState := COMM_STATE_ERROR;
    END_IF;

    // Pack outgoing data
    PackOutgoingData;

    // Communication state machine
    CASE CommState OF
        COMM_STATE_OFF:
            fb_EIPCyclic.enable := FALSE;
            IF Initialized THEN
                CommState := COMM_STATE_ON;
            END_IF;

        COMM_STATE_ON:
            fb_EIPCyclic.enable := TRUE;
            IF NOT Initialized THEN // Just provides a way to manually stop communication for debugging
                CommState := COMM_STATE_OFF;
            END_IF;

        COMM_STATE_ERROR:
            IF gMachine.Cmd.ErrorReset THEN
                // No error reset on this function block
                // Just disable and re-enable
                fb_EIPCyclic.enable := FALSE;
                CommState := COMM_STATE_OFF;
            END_IF;
    END_CASE;

    // Call communication function block cyclicall
    fb_EIPCyclic(handle := InitHandle);

    // Unpack received data
    UnpackIncomingData;

END_PROGRAM

PROGRAM _EXIT

    // Stop communication and free up resources
    // This must be called in the Exit routine
    fb_EIPExit.enable := TRUE;
    fb_EIPExit.handle := InitHandle;
    fb_EIPExit();

END_PROGRAM
```

#### Types.typ - Local data types
```iecst
(***************************************************************************************
 * EipComm task local types and enumerations
 *
 * These datatypes and enums are local to the EipComm task and are used for
 * EtherNet/IP communication
 *
 * File: EipComm/Types.typ
 * Created: 2025-03-11
 *
 * Authors:
 *  Marcus Mangel, B&R Industrial Automation
 *
***************************************************************************************)

TYPE
    CommState_enum :
        ( (*State of the communication program*)
        COMM_STATE_OFF, (*Communication is inactive*)
        COMM_STATE_ON, (*Communication is active*)
        COMM_STATE_ERROR (*There is an error. Communication is inactive*)
        );
END_TYPE

(*Communicated Data*)

TYPE
    IO_type :     STRUCT  (*Data communicated to external controller*)
        In : IO_In_type; (*Data from external controller (Output Assembly)*)
        Out : IO_Out_type; (*Data to external controller (Input Assembly)*)
    END_STRUCT;
    IO_In_type :     STRUCT  (*Data from external controller (Output Assembly)*)
        SystemEnable : BOOL; (*Command: Power all Sections*)
        SystemErrorReset : BOOL; (*Command: Global error reset*)
        TargetReleaseToTarget : DINT; (*Command: Release the Shuttle at the Target to a new Target. Bit packed (bit position = Source Target #)*)
        TargetReleaseToOffset : DINT; (*Command: Release the Shuttle to a Target with an Offset. Bit packed (bit position = Source Target #)*)
        TargetDestinationTarget : ARRAY[0..31]OF SINT; (*Parameter: Destination Target for the ReleaseToTarget command*)
        TargetReleaseDirection : ARRAY[0..31]OF INT; (*Parameter: Direction of Release. 0=CW, 1=CCW. Source Target# = Array Position. ARRAY SIZE MUST MATCH DEFINITION IN .DAT FILE*)
        TargetReleaseAccel : ARRAY[0..31]OF REAL; (*Parameter: Acceleration [m/s^2] for Release commands (Source Target# = Array Position). ARRAY SIZE MUST MATCH DEFINITION IN .DAT FILE*)
        TargetReleaseVelocity : ARRAY[0..31]OF REAL; (*Parameter: Velocity [mm/s] for Release commands (Source Target# = Array Position). ARRAY SIZE MUST MATCH DEFINITION IN .DAT FILE*)
        TargetReleaseOffset : ARRAY[0..31]OF REAL; (*Parameter: Absolute position offset from Target [mm]. (Source Target# = Array Position). ARRAY SIZE MUST MATCH DEFINITION IN .DAT FILE*)
    END_STRUCT;
    IO_Out_type :     STRUCT  (*Data to external controller (Input Assembly)*)
        SystemEnabled : BOOL; (*Status: All sections are Enabled*)
        SystemDisabled : BOOL; (*Status: All sections are Disabled*)
        SystemReadyToEnable : BOOL; (*Status: System is ready to Enable*)
        SystemFaultPresent : BOOL; (*Status: System is reporting a Fault*)
        SystemWarningPresent : BOOL; (*Status: System is reporting a Warning*)
        ProgramError : BOOL; (*Status: gMachine.Status.Error*)
        SystemFaults : DINT; (*Status: System Fault bits*)
        SystemWarnings : DINT; (*Status: System Warning bits*)
        TargetError : DINT; (*Status: A Target control function block is reporting an error. Bit packed (bit position = Target #)*)
        ShuttleError : DINT; (*Status: A Shuttle control function block is reporting an error. Bit packed (bit position = Shuttle #)*)
        TargetShuttlePresent : DINT; (*Status: A Shuttle has arrived at the Target. Bit packed (bit position = Target #)*)
        SystemSectionCount : INT; (*Status: # of configured Sections (only read once on Enable)*)
        SystemShuttleCount : INT; (*Status: # of Shuttles currently on the system (read Cyclically)*)
        SectionError : SINT; (*Status: Section # reporting a Fault*)
        SectionWarning : SINT; (*Status: Section # reporting a Warning*)
        TargetShuttleID : ARRAY[0..31]OF SINT; (*Status: ID of the Shuttle at the Target (Target# = Array Position). ARRAY SIZE MUST MATCH DEFINITION IN .DAT FILE*)
        TargetShuttleCount : ARRAY[0..31]OF SINT; (*Status: Number of Shuttles at the Target (Target# = Array Position). ARRAY SIZE MUST MATCH DEFINITION IN .DAT FILE*)
    END_STRUCT;
END_TYPE
```

#### Variables.var - Local variables
```iecst
(***************************************************************************************
 * EipComm task local variables
 *
 * These variables are local to the EipComm task and are used for
 * EtherNet/IP communication
 *
 * File: EipComm/Variables.var
 * Created: 2025-03-11
 *
 * Authors:
 *  Marcus Mangel, B&R Industrial Automation
 *
***************************************************************************************)
VAR
    CommState : CommState_enum; (*State of the communication program*)
    IO : IO_type; (*Data communicated via EtherNet/IP*)
    StationStatus : UDINT; (*Communication status data. See .dat file*)
    TaskIsSimulated : BOOL; (*If true, Input data will be ignored (allows setting via the Watch window)*)
    Initialized : BOOL; (*EIPInit block sucessfully initialized the interface in the INIT program*)
    InitHandle : UDINT; (*Handle provided by EIPInit*)
    InitExitStatus : STRING[80]; (*Exit Status provided by EIPInit. Contains error information*)
    i : USINT;
    UserLogArguments : UserLogFormatType; (*Arguments used in Logger messages (UserLog library)*)
END_VAR
(*Function Blocks*)
VAR
    fb_EIPInit : EIPInit; (*Initializes communication. Call in INIT*)
    fb_EIPCyclic : EIPCyclic; (*Cyclically performs communication. Call in CYCLIC*)
    fb_EIPExit : EIPExit; (*Shuts down communication. Call in EXIT*)
END_VAR
```

#### IO.st
```iecst
(***************************************************************************************
 * EtherNet/IP Communication Data (IO) Processing Actions
 *
 * File: EipComm/IO.st
 * Created: 2026-06-17
 *
 * Authors:
 *  Marcus Mangel, B&R Industrial Automation
 *
***************************************************************************************)

// Packs data to be transmitted over Ethernet/IP
// Arrays of BOOLs are not allowed, so these must be packed into DINTs
// Arrays of other datatypes need a fixed sized defined in the .dat file
// so data will be copied into these arrays
ACTION PackOutgoingData:

    // Copy System values directly
    IO.Out.SystemEnabled := gSuperTrak.System.Info.SectionsEnabled;
    IO.Out.SystemDisabled := gSuperTrak.System.Info.SectionsDisabled;
    IO.Out.SystemReadyToEnable := gSuperTrak.System.Status.Ready;
    IO.Out.SystemFaultPresent := gSuperTrak.System.Info.FaultPresent;
    IO.Out.SystemFaults := gSuperTrak.System.Info.Faults;
    IO.Out.SystemWarningPresent := gSuperTrak.System.Info.WarningPresent;
    IO.Out.SystemWarnings := gSuperTrak.System.Info.Warnings;
    IO.Out.SectionError := gSuperTrak.Sections.Status.SectionError;
    IO.Out.SectionWarning := gSuperTrak.Sections.Status.SectionWarning;
    IO.Out.ProgramError := gMachine.Status.Error; // In External Control mode, this is just feedback that an StCom block is errored out
    IO.Out.SystemSectionCount := gSuperTrak.System.Info.SectionCount;
    IO.Out.SystemShuttleCount := gSuperTrak.System.Info.ShuttleCount;

    // Loop through all possible Target values
    // If target numbers > 32 are used, the communication
    // definitions must be changed
    FOR i := 1 TO 32 DO
        IF i > ST_TARGET_MAX THEN
            EXIT;
        ELSE
            // Status: Shuttle Present. Pack into a DINT bitwise
            IF gSuperTrak.Target[i].Status.ShuttlePresent THEN
                IO.Out.TargetShuttlePresent := BIT_SET(IO.Out.TargetShuttlePresent, i-1);
            ELSE
                IO.Out.TargetShuttlePresent := BIT_CLR(IO.Out.TargetShuttlePresent, i-1);
            END_IF;

            // Status: Shuttle ID. Copy into a fixed-size array
            IO.Out.TargetShuttleID[i-1] := gSuperTrak.Target[i].Status.ShuttleID;

            // Status: Shuttle Count. Copy into a fixed-size array
            IO.Out.TargetShuttleCount[i-1] := gSuperTrak.Target[i].Status.ShuttleCount;

            // Status: Error on StTargetExt function block
            IF gSuperTrak.Target[i].Status.Error THEN
                IO.Out.TargetError := BIT_SET(IO.Out.TargetError, i-1);
            ELSE
                IO.Out.TargetError := BIT_CLR(IO.Out.TargetError, i-1);
            END_IF;
        END_IF;
    END_FOR;

    // Loop through all possible Shuttle values
    // If shuttle numbers > 32 are used, the communication
    // definitions must be changed
    FOR i := 1 TO 32 DO
        IF i > ST_SHUTTLE_MAX THEN
            EXIT;
        ELSE
            // Status: Error on StPallet function block
            IF gSuperTrak.Shuttle[i].Status.Error THEN
                IO.Out.ShuttleError := BIT_SET(IO.Out.ShuttleError, i-1);
            ELSE
                IO.Out.ShuttleError := BIT_CLR(IO.Out.ShuttleError, i-1);
            END_IF;
        END_IF;
    END_FOR;

END_ACTION

// Unpacks data received from Ethernet/IP
// Arrays of BOOLs are not allowed, so these must be unpacked from DINTs
// Arrays of other datatypes need a fixed sized defined in the .dat file
// so data will be copied from these arrays
ACTION UnpackIncomingData:

    // Don't try to read data if the task is being simulated
    // This will allow setting gSuperTrak members from the Watch window
    // Set TaskIsSimulated False to establish a real EthIP connection to ARSim
    IF TaskIsSimulated THEN
        RETURN;
    END_IF;

    // Copy System values directly
    gSuperTrak.System.Cmd.PowerAllSections := IO.In.SystemEnable;
    gMachine.Cmd.ErrorReset := IO.In.SystemErrorReset;

    // Loop through all possible Target values
    // If target numbers > 32 are used, the communication
    // definitions must be changed
    FOR i := 1 TO 32 DO
        IF i > ST_TARGET_MAX THEN
            EXIT;
        ELSE
            // Command: Release To Target. Unpack from a DINT bitwise
            gSuperTrak.Target[i].Cmd.Release.ReleaseToTarget := BIT_TST(IO.In.TargetReleaseToTarget, i-1);

            // Command: Release To Offset. Unpack from a DINT bitwise
            gSuperTrak.Target[i].Cmd.Release.ReleaseToOffset := BIT_TST(IO.In.TargetReleaseToOffset, i-1);

            // Parameter: Destination Target. Copy out of a fixed-size array
            gSuperTrak.Target[i].Par.Release.DestinationTarget := IO.In.TargetDestinationTarget[i-1];

            // Parameter: Release Acceleration. Copy out of a fixed-size array
            gSuperTrak.Target[i].Par.Release.Acceleration := IO.In.TargetReleaseAccel[i-1];

            // Parameter: Release Velocity. Copy out of a fixed-size array
            gSuperTrak.Target[i].Par.Release.Velocity := IO.In.TargetReleaseVelocity[i-1];

            // Parameter: Release Direction. Copy out of a fixed-size array
            gSuperTrak.Target[i].Par.Release.Direction := IO.In.TargetReleaseDirection[i-1];

            // Parameter: Release Target Offset. Copy out of a fixed-size array
            gSuperTrak.Target[i].Par.Release.TargetOffset := IO.In.TargetReleaseOffset[i-1];
        END_IF;
    END_FOR;

END_ACTION
```

#### Action.st - not listed in the package file held
```iecst
// Packs data to be transmitted over Ethernet/IP
// This is to avoid sending the entire gSuperTrak structure
// Arrays of BOOLs are not allowed
ACTION PackOutgoingData:

    // Loop through all possible target values
    // If target numbers > 31 are used, the communication
    // definitions must be changed
    FOR i := 1 TO 31 DO
        IF i > ST_TARGET_MAX THEN
            EXIT;
        ELSE
            // Set data for ShuttleInPosition
            IF gSuperTrak.Target[i].Status.ShuttleInPosition THEN
                Target_ShuttleAtTarget := BIT_SET(Target_ShuttleAtTarget, i);
            ELSE
                Target_ShuttleAtTarget := BIT_CLR(Target_ShuttleAtTarget, i);
            END_IF;

            // Set data for Shuttle Number at Target
            Target_ShuttleNumber[i] := gSuperTrak.Target[i].Status.ShuttleID;

            // Set data for Shuttle Count
            Target_ShuttleCount[i] := gSuperTrak.Target[i].Status.ShuttleCount;
        END_IF;
    END_FOR;

END_ACTION

// Unpacks data received from Ethernet/IP
// This is to avoid sending the entire gSuperTrak structure
// Arrays of BOOLs are not allowed
ACTION UnpackIncomingData:

    // Loop through all possible target values
    // If target numbers > 31 are used, the communication
    // definitions must be changed
    FOR i := 1 TO 31 DO
        IF i > ST_TARGET_MAX THEN
            EXIT;
        ELSE
            // Set data for Next Destination
            gSuperTrak.Target[i].Par.Release.DestinationTarget := Target_NextDestination[i];
            gSuperTrak.Target[i].Par.Release.Velocity := gMachine.Par.Velocity;
            gSuperTrak.Target[i].Par.Release.Acceleration := gMachine.Par.Acceleration;
            gSuperTrak.Target[i].Par.Release.Direction := gSuperTrak.System.Par.GlobalDirection;

            // Set data for Release
            gSuperTrak.Target[i].Cmd.Release.ReleaseToTarget := BIT_TST(Target_Release, i);
        END_IF;
    END_FOR;

END_ACTION
```

### Data object Logical/Source/EthIP/ethIPcon (Simple) - Configuration Data Object for the EthernetIP Communication

#### ethIPcon.dat
```
"#OWNIP=192.168.1.100"
"#OWNINTERFACE=IF3"
"#STATION=PLC"
"#STATIONIP=192.168.1.1"
"#STATIONSTATUS=EipComm:StationStatus"
"#CONNAME=Connection1"
"#CONDIR=BOTH"
"#CONRPI=10"

"#INPUTASSEMBLY=Assem1"
"EipComm:IO.Out.SystemEnabled, BOOL"
"EipComm:IO.Out.SystemDisabled, BOOL"
"EipComm:IO.Out.SystemReadyToEnable, BOOL"
"EipComm:IO.Out.SystemFaultPresent, BOOL"
"EipComm:IO.Out.SystemWarningPresent, BOOL"
"EipComm:IO.Out.SystemSectionCount, INT"
"EipComm:IO.Out.SystemShuttleCount, INT"
"EipComm:IO.Out.SystemFaults, DINT"
"EipComm:IO.Out.SystemWarnings, DINT"
"EipComm:IO.Out.TargetShuttlePresent, DINT"
"EipComm:IO.Out.TargetShuttleID, SINT, 32"
"EipComm:IO.Out.TargetShuttleCount, SINT, 32"

"#OUTPUTASSEMBLY=Assem2"
"EipComm:IO.In.SystemEnable, BOOL"
"EipComm:IO.In.SystemErrorReset, BOOL"
"EipComm:IO.In.TargetReleaseToTarget, DINT"
"EipComm:IO.In.TargetReleaseToOffset, DINT"
"EipComm:IO.In.TargetDestinationTarget, SINT, 32"
"EipComm:IO.In.TargetReleaseDirection, INT, 32"
"EipComm:IO.In.TargetReleaseAccel, REAL, 32"
"EipComm:IO.In.TargetReleaseVelocity, REAL, 32"
"EipComm:IO.In.TargetReleaseOffset, REAL, 32"
```

- SuperTrak.L5X - Allen Bradley import file (not shown)

### ReadMe.txt - EtherNet/IP Communication Instructions
```
To establish EtherNet/IP Communication between the B&R SuperTrak Controller PC and an Allen Bradley PLC:

B&R Side
1. Enable the EipComm task in the Software Configuration (Cpu.sw)
2. Modify the IP addresses in the ethIPcon.dat data file. #OWNIP refers to the B&R PC's IP address and #STATIONIP refers to the AB PLC's IP address
3. Change the #OWNINTERFACE if you're using a different ETH interface than the default (IF3/ETH1)
4. After all modifications are complete, build and transfer the Automation Studio project to the B&R controller
5. Restart the B&R controller if it did not automatically restart after the transfer

Allen Bradley Side:
1. Use "Import Program" to import the SuperTrak.L5X file. This file includes two UDTs (ST_EthIP_Input and ST_EthIP_Output), two controller tags (SuperTrak_In and SuperTrak_Out), and a copy program (SuperTrak) that moves data between the Generic Ethernet module and the controller tags
    The UDTs define the typed byte layout of the input and output assemblies
    The controller tags (SuperTrak_In / SuperTrak_Out) hold the decoded data exchanged with the B&R controller; reference these in your application logic
2. Add a Generic Ethernet module to the Allen Bradley project. Use the following settings:
    Name: Connection1
    Comm Format: Data - SINT
    IP Address: match #OWNIP from the .dat file
    Input Assembly Instance/Size: 101/96
    Output Assembly Instance/Size: 102/492
    Configuration Assembly Instance/Size: 100/400
    RPI: 10 ms
3. Schedule the copy program to run at least every 5ms (at least twice as fast as the RPI). Each scan it copies Connection1:I -> SuperTrak_In and SuperTrak_Out -> Connection1:O
    Note: the copy program references the module tags, so the module in step 2 must be named Connection1 (otherwise update the CPS operands). Verify the routine after adding the module
4. Download the Allen Bradley project to the PLC and start the program. The Generic Ethernet module should be Running with no faults
5. In your application logic, read status from SuperTrak_In.* and write commands to SuperTrak_Out.*. Do not use the raw Connection1:I / Connection1:O tags directly
```

### Package Logical/Source/MachMgr/STSystem - 1100 StCom system control

### STSystem.typ
```iecst
TYPE
	STSystemInterfaceType : 	STRUCT  (*Program interface*)
		Cmd : STSystemInterfaceCmdType;
		Status : STSystemInterfaceStatusType;
		Info : STSystemInterfaceInfoType;
	END_STRUCT;
	STSystemInterfaceCmdType : 	STRUCT  (*Interface commands*)
		Start : BOOL;
		Run : BOOL;
		Stop : BOOL;
		Reset : BOOL;
	END_STRUCT;
	STSystemInterfaceStatusType : 	STRUCT  (*Interface command response*)
		Busy : BOOL;
		Ready : BOOL;
		Running : BOOL;
		Stopped : BOOL;
		Error : BOOL;
		ErrorID : DINT;
	END_STRUCT;
	STSystemInterfaceInfoType : 	STRUCT  (*Interface information*)
		WarningPresent : BOOL; (*One or more system warnings are active*)
		Warnings : UDINT; (*System warning bits*)
		FaultPresent : BOOL; (*One or more system faults are active*)
		Faults : UDINT; (*System fault bits*)
		SectionsEnabled : BOOL; (*All sections enabled*)
		SectionsDisabled : BOOL; (*All sections disabled*)
	END_STRUCT;
END_TYPE
```

### STSystem.var
```iecst
VAR
	gSTSystem : STSystemInterfaceType;
	gSTSystemLink : StLinkType;
END_VAR
```

### Program Logical/Source/MachMgr/MachMgr

#### Main.st
```iecst
PROGRAM _INIT

	gSTSystem;

END_PROGRAM

PROGRAM _CYCLIC

END_PROGRAM

PROGRAM _EXIT

END_PROGRAM
```

### Package Logical/UserFiles - Transfer contents to USER partition

- ST_7005.dat (binary file, 704 bytes)
### Global.var - not listed in the package file held
```iecst
VAR
	gStLink : StLinkType;
END_VAR
```

### Program Logical/STCyclic

#### Variables.var
```iecst
(*Control interface*)
VAR
	ControlData : ARRAY[0..499] OF USINT;
	StatusData : ARRAY[0..499] OF USINT;
	ControlInterface : SuperTrakControlInterface_t;
END_VAR
(*Service channel*)
VAR
	PLCInterfaceRevision : UINT;
	RequestData : ARRAY[0..127] OF USINT;
	ResponseData : ARRAY[0..127] OF USINT;
	ServiceChannel : ServiceChannel_t;
	RequestHeader : REFERENCE TO ServiceChannelHeader_t;
	ResponseHeader : REFERENCE TO ServiceChannelHeader_t;
END_VAR
(*StCom system control*)
VAR
	ControlSystem : StControl;
	SystemParameters : StControlParType;
END_VAR
```

#### Main.st
```iecst
PROGRAM _INIT

	// Initialize SuperTrak, set configuration path
	SuperTrakInit('/DEVICE=USER_PATH\SuperTrak\Configuration', '127.0.0.1', 'IF3,IF4');

	// Set PLC interface to revision 0 for StCom
	PLCInterfaceRevision := 0;
	SuperTrakServChanWrite(0, stPAR_PLC_IF_REVISION, 0, 1, ADR(PLCInterfaceRevision), SIZEOF(PLCInterfaceRevision));

	// Initialize StCom system parameters
	SystemParameters.NrOfCommands := 48;
	SystemParameters.NrOfSections := 4;
	SystemParameters.NrOfTargets := 4;
	SystemParameters.NrOfPallets := 4;
	ControlSystem.Enable := TRUE;

	// Initialize service channel identifier for StCom
	ServiceChannel.channelId := 1;

END_PROGRAM

PROGRAM _CYCLIC

	// Process control and status data of PLC interface for StCom
	ControlInterface.pControl := ADR(ControlData);
	ControlInterface.pStatus := ADR(StatusData);
	ControlInterface.controlSize := SIZEOF(ControlData);
	ControlInterface.statusSize := SIZEOF(StatusData);

	// Process control data before SuperTrak cyclic and status data after
	SuperTrakProcessControl(0, ControlInterface);
	SuperTrakCyclic1();
	SuperTrakProcessStatus(0, ControlInterface);

	// Call StCom system
	// This function block receives commands from other StCom function blocks
	// The commands are processed in the PLC interface
	ControlSystem.StLink := ADR(gStLink);
	ControlSystem.Parameters := ADR(SystemParameters);
	ControlSystem.StCtrlData := ADR(ControlData);
	ControlSystem.StCtrlDataSize := SIZEOF(ControlData);
	ControlSystem.StStatData := ADR(StatusData);
	ControlSystem.StStatDataSize := SIZEOF(StatusData);
	ControlSystem.StServChRequestData := ADR(RequestData);
	ControlSystem.StServChRequestDataSize := SIZEOF(RequestData);
	ControlSystem.StServChResponseData := ADR(ResponseData);
	ControlSystem.StServChResponseDataSize := SIZEOF(ResponseData);
	ControlSystem();

	// Call service channel
	// This is used for a short amount of time to configure the PLC interface for StCom
	ServiceChannel.pRequestHeader := ADR(RequestData);
	ServiceChannel.pResponseHeader := ADR(ResponseData);
	ServiceChannel.pRequestValues := ADR(RequestData) + SIZEOF(ServiceChannelHeader_t);
	ServiceChannel.pResponseValues := ADR(ResponseData) + SIZEOF(ServiceChannelHeader_t);
	ServiceChannel.requestBufferSize := SIZEOF(RequestData) - SIZEOF(ServiceChannelHeader_t);
	ServiceChannel.responseBufferSize := SIZEOF(ResponseData) - SIZEOF(ServiceChannelHeader_t);
	RequestHeader ACCESS ADR(RequestData);
	ResponseHeader ACCESS ADR(ResponseData);

	IF ServiceChannel.state = scSTATE_RECV AND RequestHeader.sequence <> ResponseHeader.sequence THEN
		ServiceChannel.requestSequence := RequestHeader.sequence;
		ServiceChannel.state := scSTATE_EXEC;

	ELSIF ServiceChannel.state = scSTATE_EXEC OR ServiceChannel.state = scSTATE_WAIT THEN
		SuperTrakServiceChannel(ServiceChannel);

	ELSIF ServiceChannel.state = scSTATE_SEND THEN
		ServiceChannel.state := scSTATE_RECV;
	END_IF

END_PROGRAM

PROGRAM _EXIT

	SuperTrakExit();

END_PROGRAM
```

### Package Logical/Tasks/MachMgr - Machine manager

### Program Logical/Tasks/MachMgr/MachMgr (IEC) - Machine manager

#### Variables.var
```iecst
VAR
	Index : USINT;
END_VAR
```

#### Main.st
```iecst
PROGRAM _INIT

	// Assign section number to each element
	FOR Index := 1 TO ST_SECTION_MAX DO
		gSTSection.Par.Section[Index] := Index;
	END_FOR

END_PROGRAM

PROGRAM _CYCLIC

	// Enable section function blocks when the system function block is active
	gSTSection.Cmd.Enable := gSTSystem.Status.Ready;

END_PROGRAM

PROGRAM _EXIT

END_PROGRAM
```

### Package Logical/Tasks/MachMgr/STCyclic - SuperTrak cyclic update

### STCyclic.typ - Global types
```iecst
TYPE
	STCyclicInterfaceType : 	STRUCT  (*Interface structure*)
		Status : STCyclicInterfaceStatusType; (*Status structure*)
	END_STRUCT;
	STCyclicInterfaceStatusType : 	STRUCT  (*Status structure*)
		Reference : STCyclicInterfaceReferenceType;
	END_STRUCT;
	STCyclicInterfaceReferenceType : 	STRUCT  (*Status structure*)
		ControlDataAddress : UDINT;
		ControlDataSize : UDINT;
		StatusDataAddress : UDINT;
		StatusDataSize : UDINT;
		RequestDataAddress : UDINT;
		RequestDataSize : UDINT;
		ResponseDataAddress : UDINT;
		ResponseDataSize : UDINT;
	END_STRUCT;
END_TYPE
```

### STCyclic.var - Global variables
```iecst
VAR
	gSTCyclicReference : STCyclicReferenceType;
END_VAR
```

### Program Logical/Tasks/MachMgr/STCyclic/STCyclic (IEC) - SuperTrak cyclic update and StCom control

#### Log.var
```iecst
VAR
	FirstScan : BOOL := TRUE; (*Log timestamp of first scan*)
	PreviousStComActive : BOOL; (*Montior for change in StControl active status*)
	PreviousServiceChannelState : USINT; (*Montior for change in service channel processing states*)
	Values : UserLogFormatType; (*Runtime values for formatted log messages*)
END_VAR
```

#### Variables.var
```iecst
(*PLC interface*)
VAR
	ControlData : ARRAY[0..499] OF USINT; (*Raw input data to PLC interface used for StCom*)
	StatusData : ARRAY[0..499] OF USINT; (*Raw output data from PLC interface used for StCom*)
	PLCInterfaceParameters : SuperTrakControlInterface_t; (*PLC interface data parameters*)
END_VAR
(*Service channel*)
VAR
	PLCInterfaceRevision : UINT; (*Revision number 0 required for StCom*)
	RequestData : ARRAY[0..127] OF USINT; (*Raw service channel input data used for StCom*)
	ResponseData : ARRAY[0..127] OF USINT; (*Raw service channel output data used for StCom*)
	ServiceChannel : ServiceChannel_t; (*Service channel instance interface*)
	RequestHeader : REFERENCE TO ServiceChannelHeader_t; (*Pointer to header in raw service channel input data*)
	ResponseHeader : REFERENCE TO ServiceChannelHeader_t; (*Pointer to header in raw sercive channel output data*)
END_VAR
```

#### Log.st
```iecst
ACTION LogStComServiceChannel:

	// Read Section Count 1080
	// Read System Name 1053
	// Read Enable Signal Source 1057
	// Write PLC Interface Options 1430
	// Write PLC Interface Section Count 1432
	// Write PLC Interface Target Count 1434
	// Write PLC Interface Command Count 1436
	// Write Parameter Save Function 971

	IF ServiceChannel.state = scSTATE_EXEC AND ServiceChannel.state <> PreviousServiceChannelState THEN
		Values.i[0] := RequestHeader.task;
		Values.i[1] := RequestHeader.param;
		Values.i[2] := RequestHeader.section;
		Values.i[3] := RequestHeader.count;
		UserLogAdvanced(USERLOG_SEVERITY_INFORMATION, 100, 'Service Channel request execution, task %i, parameter %i, Section %i, Count %i', Values);
	END_IF

	PreviousServiceChannelState := ServiceChannel.state;

END_ACTION
```

#### Main.st
```iecst
PROGRAM _INIT

	// Initialize SuperTrak, set configuration path
	SuperTrakInit('/DEVICE=USER_PATH\SuperTrak\Configuration', '127.0.0.1', 'IF3,IF4');

	// Set PLC interface to revision 0 for StCom
	PLCInterfaceRevision := 0;
	SuperTrakServChanWrite(0, stPAR_PLC_IF_REVISION, 0, 1, ADR(PLCInterfaceRevision), SIZEOF(PLCInterfaceRevision));

	// Initialize service channel identifier for StCom
	ServiceChannel.channelId := 1;

END_PROGRAM

PROGRAM _CYCLIC

	// Process control and status data of PLC interface for StCom
	PLCInterfaceParameters.pControl := ADR(ControlData);
	PLCInterfaceParameters.pStatus := ADR(StatusData);
	PLCInterfaceParameters.controlSize := SIZEOF(ControlData);
	PLCInterfaceParameters.statusSize := SIZEOF(StatusData);

	// Process control data before SuperTrak cyclic and status data after
	SuperTrakProcessControl(0, PLCInterfaceParameters);
	SuperTrakCyclic1();
	SuperTrakProcessStatus(0, PLCInterfaceParameters);

	// Call service channel
	// This is used for a short amount of time to configure the PLC interface for StCom
	ServiceChannel.pRequestHeader := ADR(RequestData);
	ServiceChannel.pResponseHeader := ADR(ResponseData);
	ServiceChannel.pRequestValues := ADR(RequestData) + SIZEOF(ServiceChannelHeader_t);
	ServiceChannel.pResponseValues := ADR(ResponseData) + SIZEOF(ServiceChannelHeader_t);
	ServiceChannel.requestBufferSize := SIZEOF(RequestData) - SIZEOF(ServiceChannelHeader_t);
	ServiceChannel.responseBufferSize := SIZEOF(ResponseData) - SIZEOF(ServiceChannelHeader_t);
	RequestHeader ACCESS ADR(RequestData);
	ResponseHeader ACCESS ADR(ResponseData);

	// StCom has access to request and response data
	// The SuperTrakServiceChannel function is called when the sequence count increments
	// See the SuperTrak library help for SuperTrakServiceChannel
	IF ServiceChannel.state = scSTATE_RECV AND RequestHeader.sequence <> ResponseHeader.sequence THEN
		ServiceChannel.requestSequence := RequestHeader.sequence;
		ServiceChannel.state := scSTATE_EXEC;

	ELSIF ServiceChannel.state = scSTATE_EXEC OR ServiceChannel.state = scSTATE_WAIT THEN
		SuperTrakServiceChannel(ServiceChannel);

	ELSIF ServiceChannel.state = scSTATE_SEND THEN
		ServiceChannel.state := scSTATE_RECV;
	END_IF

	// Share data access to StCom's StControl
	Interface.Status.Reference.ControlDataAddress := ADR(ControlData);
	Interface.Status.Reference.ControlDataSize := SIZEOF(ControlData);
	Interface.Status.Reference.StatusDataAddress := ADR(StatusData);
	Interface.Status.Reference.StatusDataSize := SIZEOF(StatusData);
	Interface.Status.Reference.RequestDataAddress := ADR(RequestData);
	Interface.Status.Reference.RequestDataSize := SIZEOF(RequestData);
	Interface.Status.Reference.ResponseDataAddress := ADR(ResponseData);
	Interface.Status.Reference.ResponseDataSize := SIZEOF(ResponseData);

	// Log service channel requests
	LogStComServiceChannel;

END_PROGRAM

PROGRAM _EXIT

	SuperTrakExit();

END_PROGRAM
```

### Package Logical/Tasks/MachMgr/STSystem - 1100 StCom system control

### STSystem.typ
```iecst
TYPE
	STSystemInterfaceType : 	STRUCT
		Cmd : STSystemInterfaceCmdType;
		Status : STSystemInterfaceStatusType;
		Info : STSystemInterfaceInfoType;
	END_STRUCT;
	STSystemInterfaceCmdType : 	STRUCT
		Start : BOOL;
		Run : BOOL;
		Stop : BOOL;
		Reset : BOOL;
	END_STRUCT;
	STSystemInterfaceStatusType : 	STRUCT
		Busy : BOOL;
		Ready : BOOL;
		Running : BOOL;
		Stopped : BOOL;
		Error : BOOL;
		ErrorID : DINT;
	END_STRUCT;
	STSystemInterfaceInfoType : 	STRUCT
		WarningPresent : BOOL; (*One or more system warnings are active*)
		Warnings : UDINT; (*System warning bits*)
		FaultPresent : BOOL; (*One or more system faults are active*)
		Faults : UDINT; (*System fault bits*)
		SectionsEnabled : BOOL; (*All sections enabled*)
		SectionsDisabled : BOOL; (*All sections configured in the PLC interface are disabled*)
	END_STRUCT;
END_TYPE
```

### STSystem.var
```iecst
VAR
	gSTSystemLink : StLinkType;
END_VAR
```

### Program Logical/Tasks/MachMgr/STSystem/STSystem (IEC)

#### Main.st - Init, cyclic, exit code
```iecst
PROGRAM _INIT

	SystemParameters.NrOfCommands := 24;
	SystemParameters.NrOfSections := 4;
	SystemParameters.NrOfTargets := 4;
	SystemParameters.NrOfPallets := 4;

	Timeout.PT := T#500ms;

END_PROGRAM

PROGRAM _CYCLIC

	// Read global inputs
	Interface.Cmd := gSTSystem.Cmd;

	// State control
	CASE State OF
		STATE_OFF:
			IF StartTrigger.Q THEN
				State := STATE_INITIALIZE;
			END_IF

		STATE_INITIALIZE:
			// Enable once and never disabled
			ControlSystem.Enable := TRUE;

			IF ControlSystem.Active THEN
				State := STATE_IDLE;

			ELSIF ControlSystem.Error THEN
				Interface.Status.ErrorID := ControlSystem.StatusID;
				State := STATE_ERROR;

			ELSIF Timeout.Q THEN
				Interface.Status.ErrorID := -1;
				State := STATE_ERROR;
			END_IF

		STATE_IDLE:
			IF ControlSystem.SectionsEnabled THEN
				UserLogBasic(USERLOG_SEVERITY_WARNING, 1102, 'Sections enabled by alternative source');
				State := STATE_EXECUTE;

			ELSIF RunTrigger.Q THEN
				State := STATE_STARTING;

			ELSIF ControlSystem.Error THEN
				Interface.Status.ErrorID := ControlSystem.StatusID;
				State := STATE_ERROR;
			END_IF

		STATE_STARTING:
			ControlSystem.EnableAllSections := TRUE;

			IF ControlSystem.SectionsEnabled THEN
				State := STATE_EXECUTE;

			ELSIF ControlSystem.Error THEN
				Interface.Status.ErrorID := ControlSystem.StatusID;
				State := STATE_ERROR;

			ELSIF Timeout.Q THEN
				Interface.Status.ErrorID := -1;
				State := STATE_ERROR;
			END_IF

		STATE_EXECUTE:
			IF Interface.Info.SectionsDisabled THEN
				UserLogBasic(USERLOG_SEVERITY_WARNING, 1104, 'Sections disabled by alternative source');
				ControlSystem.EnableAllSections := FALSE;
				State := STATE_IDLE;

			ELSIF Interface.Cmd.Stop THEN
				State := STATE_STOPPING;

			ELSIF ControlSystem.Error THEN
				Interface.Status.ErrorID := ControlSystem.StatusID;
				State := STATE_ERROR;
			END_IF

		STATE_STOPPING:
			ControlSystem.EnableAllSections := FALSE;

			IF Interface.Info.SectionsDisabled THEN
				State := STATE_IDLE;

			ELSIF ControlSystem.Error THEN
				Interface.Status.ErrorID := ControlSystem.StatusID;
				State := STATE_ERROR;

			ELSIF Timeout.Q THEN
				Interface.Status.ErrorID := -1;
				State := STATE_ERROR;
			END_IF

		STATE_ERROR:
			ControlSystem.EnableAllSections := FALSE;

			IF ResetTrigger.Q THEN
				State := STATE_CLEARING;
			END_IF

		STATE_CLEARING:
			ControlSystem.ErrorReset := TRUE;
			Interface.Status.ErrorID := 0;

			IF ControlSystem.Error = FALSE THEN
				ControlSystem.ErrorReset := FALSE;
				State := STATE_OFF;

			ELSIF Timeout.Q THEN
				Interface.Status.ErrorID := -1;
				State := STATE_ERROR;
			END_IF
	END_CASE

	// Call function blocks
	ControlSystem.StCtrlData := gSTCyclicReference.ControlDataAddress;
	ControlSystem.StCtrlDataSize := gSTCyclicReference.ControlDataSize;
	ControlSystem.StStatData := gSTCyclicReference.StatusDataAddress;
	ControlSystem.StStatDataSize := gSTCyclicReference.StatusDataSize;
	ControlSystem.StServChRequestData := gSTCyclicReference.RequestDataAddress;
	ControlSystem.StServChRequestDataSize := gSTCyclicReference.RequestDataSize;
	ControlSystem.StServChResponseData := gSTCyclicReference.ResponseDataAddress;
	ControlSystem.StServChResponseDataSize := gSTCyclicReference.ResponseDataSize;
	ControlSystem.StLink := ADR(gSTSystemLink);
	ControlSystem.Parameters := ADR(SystemParameters);
	ControlSystem();

	StartTrigger.CLK := Interface.Cmd.Start;
	StartTrigger();
	RunTrigger.CLK := Interface.Cmd.Run;
	RunTrigger();
	ResetTrigger.CLK := Interface.Cmd.Reset;
	ResetTrigger();

	Timeout.IN := Interface.Status.Busy;
	Timeout();

	// Process outputs
	CollectSectionStatuses;
	Interface.Info.WarningPresent := ControlSystem.Info.SuperTrak.SystemWarningActive;
	Interface.Info.Warnings := ControlSystem.Info.SuperTrak.SystemWarningBits;
	Interface.Info.FaultPresent := ControlSystem.Info.SuperTrak.SystemFaultActive;
	Interface.Info.Faults := ControlSystem.Info.SuperTrak.SystemFaultBits;

	// Set status
	Interface.Status.Busy := State = STATE_INITIALIZE OR
							State = STATE_STARTING OR
							State = STATE_STOPPING OR
							State = STATE_CLEARING;
	Interface.Status.Ready := Interface.Cmd.Stop = FALSE AND State = STATE_IDLE;
	Interface.Status.Running := State = STATE_EXECUTE;
	Interface.Status.Stopped := Interface.Cmd.Stop AND State = STATE_IDLE;
	Interface.Status.Error := State = STATE_ERROR;

	// Write global outputs
	gSTSystem.Status := Interface.Status;
	gSTSystem.Info := Interface.Info;

END_PROGRAM

PROGRAM _EXIT

END_PROGRAM
```

#### Types.typ - Local types
```iecst
TYPE
	StateEnum :
		(
		STATE_OFF, (*No action, wait for start*)
		STATE_INITIALIZE, (*Enable StControl function block*)
		STATE_IDLE, (*No action, wait for run*)
		STATE_STARTING, (*Enable all sections*)
		STATE_EXECUTE, (*Running, wait for stop*)
		STATE_STOPPING, (*Disable all sections*)
		STATE_ERROR, (*An error occurred*)
		STATE_CLEARING (*Reset error*)
		);
END_TYPE
```

#### Variables.var - Local variables
```iecst
(*Control*)
VAR
	State : StateEnum;
	Interface : STSystemInterfaceType;
END_VAR
(*Function blocks*)
VAR
	StartTrigger : R_TRIG;
	RunTrigger : R_TRIG;
	ResetTrigger : R_TRIG;
	ControlSystem : StControl;
	SystemParameters : StControlParType;
	Timeout : TON;
END_VAR
(*Data*)
VAR
	SectionStatus : REFERENCE TO USINT;
	PLCInterfaceConfiguration : SuperTrakControlIfConfig_t;
	Index : UINT;
END_VAR
```

#### Log.var - not listed in the package file held
```iecst
VAR
	FirstScan : BOOL := TRUE; (*Flag first scan of cyclic*)
	PreviousActive : BOOL; (*Previous StControl Active status*)
END_VAR
```

#### Error.st - not listed in the package file held
```iecst
ACTION ThrowError:

	LogValues.i[0] := Interface.Status.ErrorID;
	LogValues.s[0] := StateName;
	UserLogAdvanced(USERLOG_SEVERITY_ERROR, 1001, 'Error %i in state %s', LogValues);

	Interface.Status.Ready := FALSE;
	Interface.Status.Running := FALSE;
	Interface.Status.Stopped := FALSE;
	Interface.Status.Error := TRUE;

	State := STATE_ERROR;

END_ACTION
```

#### Log.st - not listed in the package file held
```iecst
ACTION LogStControlActive:

	IF FirstScan THEN
		FirstScan := FALSE;
		UserLogBasic(USERLOG_SEVERITY_INFORMATION, 200, 'First scan of cyclic');
	END_IF

	IF ControlSystem.Active AND PreviousActive = FALSE THEN
		UserLogBasic(USERLOG_SEVERITY_INFORMATION, 200, 'StControl function block not active');
	END_IF
	PreviousActive := ControlSystem.Active;

END_ACTION
```

#### State.st - not listed in the package file held
```iecst
ACTION SetStateName:

	CASE State OF
		STATE_OFF: StateName := 'OFF';
		STATE_ENABLING: StateName := 'ENABLING';
		STATE_IDLE: StateName := 'IDLE';
		STATE_RUNNING: StateName := 'RUNNING';
		STATE_STOPPED: StateName := 'STOPPED';
		STATE_ERROR: StateName := 'ERROR';
		STATE_RESETTING: StateName := 'RESETTING';
		ELSE StateName := 'UNKNOWN';
	END_CASE

END_ACTION

ACTION LogStateChange:

	IF State <> PreviousState THEN
		LogValues.s[0] := PreviousStateName;
		LogValues.s[1] := StateName;
		UserLogAdvanced(USERLOG_SEVERITY_INFORMATION, 1000, 'State changed from %s to %s', LogValues);
	END_IF
	PreviousState := State;

END_ACTION
```

### Package Logical/Tasks/MachMgr/STSection - StCom section control

### STSection.typ
```iecst
TYPE
	STSectionInterfaceType : 	STRUCT
		Cmd : STSectionInterfaceCmdType;
		Par : STSectionInterfaceParType;
		Status : STSectionInterfaceStatusType;
	END_STRUCT;
	STSectionInterfaceCmdType : 	STRUCT
		Enable : BOOL;
		EnableSection : ARRAY[1..ST_SECTION_MAX]OF BOOL;
		Reset : BOOL;
	END_STRUCT;
	STSectionInterfaceParType : 	STRUCT
		Section : ARRAY[1..ST_SECTION_MAX]OF USINT;
	END_STRUCT;
	STSectionInterfaceStatusType : 	STRUCT
		Active : BOOL;
		Error : BOOL;
		SectionEnabled : ARRAY[1..ST_SECTION_MAX]OF BOOL;
	END_STRUCT;
END_TYPE
```

### STSection.var
```iecst
VAR CONSTANT
	ST_SECTION_MAX : USINT := 4;
END_VAR
VAR
	gSTSection : STSectionInterfaceType;
END_VAR
```

### Program Logical/Tasks/MachMgr/STSection/STSection

#### Variables.var
```iecst
VAR
	Interface : STSectionInterfaceType;
	SectionParameters : StSectionParType; (*Placeholder, there are no parameters for StCom's StSection function block*)
	ControlSection : ARRAY[1..ST_SECTION_MAX] OF StSection;
	Index : USINT;
END_VAR
```

#### Main.st
```iecst
PROGRAM _INIT

END_PROGRAM

PROGRAM _CYCLIC

	// Initialize common statuses, assume true/false then disqualify
	Interface.Status.Active := TRUE;
	Interface.Status.Error := FALSE;

	FOR Index := 1 TO ST_SECTION_MAX DO
		ControlSection[Index].StLink := ADR(gSTSystemLink);
		ControlSection[Index].Section := Interface.Par.Section[Index];
		// There are no function block parameters, use common address
		ControlSection[Index].Parameters := ADR(SectionParameters);
		// Enable all function blocks
		ControlSection[Index].Enable := Interface.Cmd.Enable;
		// Enable each section
		ControlSection[Index].EnableSection := Interface.Cmd.EnableSection[Index];
		// Reset all function blocks
		ControlSection[Index].ErrorReset := Interface.Cmd.Reset;
		ControlSection[Index]();

		// All sections must be active
		IF ControlSection[Index].Active = FALSE THEN
			Interface.Status.Active := FALSE;
		END_IF
		// Error if any section has error
		IF ControlSection[Index].Error THEN
			Interface.Status.Error := TRUE;
		END_IF
		Interface.Status.SectionEnabled[Index] := ControlSection[Index].SectionEnabled;
	END_FOR

END_PROGRAM

PROGRAM _EXIT

END_PROGRAM
```

### Package Logical/Tasks/MachMgr/STPosError - Force pallet position following error

### Program Logical/Tasks/MachMgr/STPosError/STPosError

#### Variables.var
```iecst
VAR CONSTANT
	PALLET_MAX : USINT := 2;
END_VAR
VAR
	PalletInfo : ARRAY[0..PALLET_MAX] OF SuperTrakPalletInfo_t;
	Index : USINT;
	SelectPalletIndex : USINT;
	TriggerSection : USINT;
	TriggerPosition : DINT;
	CreateFault : BOOL;
	CreateFaultTrigger : R_TRIG;
	PreviousPalletPosition : DINT;
	State : USINT;
END_VAR
```

#### Main.st
```iecst
PROGRAM _INIT

	TriggerSection := 3;
	TriggerPosition := 800_000;

	SelectPalletIndex := 0;

END_PROGRAM

PROGRAM _CYCLIC

	CASE State OF
		0:
			IF CreateFaultTrigger.Q THEN
				State := 10;
			END_IF

		10:
			IF SelectPalletIndex >= PALLET_MAX AND PALLET_MAX > 0 THEN
				SelectPalletIndex := PALLET_MAX - 1;
			END_IF

			SuperTrakGetPalletInfo(ADR(PalletInfo), PALLET_MAX, FALSE);
			PreviousPalletPosition := PalletInfo[SelectPalletIndex].position;

			State := 20;

		20:
			SuperTrakGetPalletInfo(ADR(PalletInfo), PALLET_MAX, FALSE);

			IF CreateFault = FALSE THEN
				State := 0;

			ELSIF PalletInfo[SelectPalletIndex].section = TriggerSection AND
				PalletInfo[SelectPalletIndex].position >= TriggerPosition AND
				PreviousPalletPosition < TriggerPosition THEN

				State := 30;
			END_IF
			PreviousPalletPosition := PalletInfo[SelectPalletIndex].position;

		30:
			SuperTrakBeginExternalControl(PalletInfo[SelectPalletIndex].palletID);

			SuperTrakPalletControl(PalletInfo[SelectPalletIndex].palletID, 1, 0, 0.0, 0.0);

			State := 40;

		40:
			State := 0;
	END_CASE

	CreateFaultTrigger.CLK := CreateFault;
	CreateFaultTrigger();

END_PROGRAM

PROGRAM _EXIT

END_PROGRAM
```

### STCyclic.typ - Global types
```iecst
TYPE
	STCyclicInterfaceType : 	STRUCT  (*Interface structure*)
		Status : STCyclicInterfaceStatusType; (*Status structure*)
	END_STRUCT;
	STCyclicInterfaceStatusType : 	STRUCT  (*Status structure*)
		Active : BOOL; (*StCom system active*)
		LinkAddress : UDINT; (*StCom StLink address*)
	END_STRUCT;
END_TYPE
```

### STCyclic.var - Global variables
```iecst
VAR
	gSTCyclic : STCyclicInterfaceType; (*Global interface*)
END_VAR
```

### Program Logical/Tasks/STCyclic/STCyclic (IEC)

#### Main.st - Init, cyclic, exit code
```iecst
PROGRAM _INIT

	// Initialize SuperTrak, set configuration path
	SuperTrakInit('/DEVICE=USER_PATH\SuperTrak\Configuration', '127.0.0.1', 'IF3,IF4');

	// Set PLC interface to revision 0 for StCom
	PLCInterfaceRevision := 0;
	SuperTrakServChanWrite(0, stPAR_PLC_IF_REVISION, 0, 1, ADR(PLCInterfaceRevision), SIZEOF(PLCInterfaceRevision));

	// Initialize StCom system parameters
	SystemParameters.NrOfCommands := 48;
	SystemParameters.NrOfSections := 4;
	SystemParameters.NrOfTargets := 4;
	SystemParameters.NrOfPallets := 4;
	ControlSystem.Enable := TRUE;

	// Initialize service channel identifier for StCom
	ServiceChannel.channelId := 1;

END_PROGRAM

PROGRAM _CYCLIC

	// Process control and status data of PLC interface for StCom
	ControlInterface.pControl := ADR(ControlData);
	ControlInterface.pStatus := ADR(StatusData);
	ControlInterface.controlSize := SIZEOF(ControlData);
	ControlInterface.statusSize := SIZEOF(StatusData);

	// Process control data before SuperTrak cyclic and status data after
	SuperTrakProcessControl(0, ControlInterface);
	SuperTrakCyclic1();
	SuperTrakProcessStatus(0, ControlInterface);

	// Call StCom system
	// This function block receives commands from other StCom function blocks
	// The commands are processed in the PLC interface
	ControlSystem.StLink := ADR(StComLink);
	ControlSystem.Parameters := ADR(SystemParameters);
	ControlSystem.StCtrlData := ADR(ControlData);
	ControlSystem.StCtrlDataSize := SIZEOF(ControlData);
	ControlSystem.StStatData := ADR(StatusData);
	ControlSystem.StStatDataSize := SIZEOF(StatusData);
	ControlSystem.StServChRequestData := ADR(RequestData);
	ControlSystem.StServChRequestDataSize := SIZEOF(RequestData);
	ControlSystem.StServChResponseData := ADR(ResponseData);
	ControlSystem.StServChResponseDataSize := SIZEOF(ResponseData);
	ControlSystem();

	// Call service channel
	// This is used for a short amount of time to configure the PLC interface for StCom
	ServiceChannel.pRequestHeader := ADR(RequestData);
	ServiceChannel.pResponseHeader := ADR(ResponseData);
	ServiceChannel.pRequestValues := ADR(RequestData) + SIZEOF(ServiceChannelHeader_t);
	ServiceChannel.pResponseValues := ADR(ResponseData) + SIZEOF(ServiceChannelHeader_t);
	ServiceChannel.requestBufferSize := SIZEOF(RequestData) - SIZEOF(ServiceChannelHeader_t);
	ServiceChannel.responseBufferSize := SIZEOF(ResponseData) - SIZEOF(ServiceChannelHeader_t);
	RequestHeader ACCESS ADR(RequestData);
	ResponseHeader ACCESS ADR(ResponseData);

	IF ServiceChannel.state = scSTATE_RECV AND RequestHeader.sequence <> ResponseHeader.sequence THEN
		ServiceChannel.requestSequence := RequestHeader.sequence;
		ServiceChannel.state := scSTATE_EXEC;

	ELSIF ServiceChannel.state = scSTATE_EXEC OR ServiceChannel.state = scSTATE_WAIT THEN
		SuperTrakServiceChannel(ServiceChannel);

	ELSIF ServiceChannel.state = scSTATE_SEND THEN
		ServiceChannel.state := scSTATE_RECV;
	END_IF

	// Share StCom link and active status
	Interface.Status.LinkAddress := ADR(StComLink);
	Interface.Status.Active := ControlSystem.Active;

	// User logging
	LogStComSystemStatus;
	LogStComServiceChannel;

END_PROGRAM

PROGRAM _EXIT

	SuperTrakExit();

END_PROGRAM
```

#### Variables.var - Local variables
```iecst
(*PLC interface*)
VAR
	ControlData : ARRAY[0..499] OF USINT; (*Raw input data to PLC interface used for StCom*)
	StatusData : ARRAY[0..499] OF USINT; (*Raw output data from PLC interface used for StCom*)
	PLCInterfaceParameters : SuperTrakControlInterface_t; (*PLC interface data parameters*)
END_VAR
(*Service channel*)
VAR
	PLCInterfaceRevision : UINT; (*Revision number 0 required for StCom*)
	RequestData : ARRAY[0..127] OF USINT; (*Raw service channel input data used for StCom*)
	ResponseData : ARRAY[0..127] OF USINT; (*Raw service channel output data used for StCom*)
	ServiceChannel : ServiceChannel_t; (*Service channel instance interface*)
	RequestHeader : REFERENCE TO ServiceChannelHeader_t; (*Pointer to header in raw service channel input data*)
	ResponseHeader : REFERENCE TO ServiceChannelHeader_t; (*Pointer to header in raw sercive channel output data*)
END_VAR
(*StCom control*)
VAR
	Interface : STCyclicInterfaceType; (*Task interface*)
	StComLink : StLinkType; (*Link for all StCom function blocks*)
	ControlStCom : StControl; (*StCom runtime manager and SuperTrak system control function block*)
	StComParameters : StControlParType; (*StControl function block parameters*)
END_VAR
```

#### Log.var
```iecst
VAR
	FirstScan : BOOL := TRUE;
	PreviousStComSystemActive : BOOL;
	PreviousServiceChannelState : USINT;
	Values : UserLogFormatType;
END_VAR
```

#### Log.st
```iecst
ACTION LogStComSystemStatus:

	IF FirstScan THEN
		FirstScan := FALSE;
		UserLogBasic(USERLOG_SEVERITY_INFORMATION, 200, 'First scan');
	END_IF

	IF ControlStCom.Active AND NOT PreviousStComActive THEN
		UserLogBasic(USERLOG_SEVERITY_INFORMATION, 210, 'StCom StSystem function block active');
	END_IF

	PreviousStComActive := ControlStCom.Active;

END_ACTION

ACTION LogStComServiceChannel:

	// Read Section Count 1080
	// Read System Name 1053
	// Read Enable Signal Source 1057
	// Write PLC Interface Options 1430
	// Write PLC Interface Section Count 1432
	// Write PLC Interface Target Count 1434
	// Write PLC Interface Command Count 1436
	// Write Parameter Save Function 971

	IF ServiceChannel.state = scSTATE_EXEC AND ServiceChannel.state <> PreviousServiceChannelState THEN
		Values.i[0] := RequestHeader.task;
		Values.i[1] := RequestHeader.param;
		Values.i[2] := RequestHeader.section;
		Values.i[3] := RequestHeader.count;
		UserLogAdvanced(USERLOG_SEVERITY_INFORMATION, 220, 'Service Channel request execution, task %i, parameter %i, Section %i, Count %i', Values);
	END_IF

	PreviousServiceChannelState := ServiceChannel.state;

END_ACTION
```

### Program Logical/TrakCyclic

#### Main.st
```iecst
PROGRAM _INIT
	SuperTrakInit('/DEVICE=USER_PATH\SuperTrak\Configuration', '127.0.0.1', 'IF3,IF4');
END_PROGRAM

PROGRAM _CYCLIC
	SuperTrakCyclic1();
END_PROGRAM

PROGRAM _EXIT
	SuperTrakExit();
END_PROGRAM
```

Listed in the project but not available here: Logical/Libraries/StHelper/Types.typ, Logical/Source/MachineMgr/STMgr/Machine.var, Logical/Source/MachineMgr/STMgr/STCyclic/STCyclic/Reference.st, Logical/Source/MachMgr/STCyclic, Logical/Source/MachMgr/STSection, Logical/Tasks/MachMgr/STSystem/STSystem/Sections.st
